// TIA Portal V20 export
// export: Created 2025-12-01T14:57:14.5855708Z, ExportSetting None, DisplayName Totally Integrated Automation Portal, DisplayVersion V20 Update 3, DisplayName TIA Portal Openness, DisplayVersion V20 Update 3, DisplayName TIA Portal Version Control Interface, DisplayVersion V20 Update 3, DisplayName STEP 7 Professional, DisplayVersion V20 Update 3, DisplayName STEP 7 Safety, DisplayVersion V20 Update 2, DisplayName WinCC Basic/Comfort/Advanced, DisplayVersion V20 Update 3, DisplayName WinCC Professional, DisplayVersion V20 Update 3, DisplayName WinCC Unified, DisplayVersion V20 Update 3
FUNCTION "FC700_JDT02ControlTracking" : Void   // FC700, LAD
{ S7_Optimized_Access := 'FALSE' }
AUTHOR : TRACKING
NAME : 20141014
VERSION : 4.0
// stored: AutoNumber false, SetENOAutomatically false
BEGIN

NETWORK
TITLE = Previo
// -----------------------------------------------------------------------
// --- Inicialializacion
// --- Borrado de la Base de Datosç

      CALL  "FC701_JDT02ControlCOM";  // Control del Puerto
      CALL  "FC706_JDT02Borrado";



NETWORK
TITLE = Control del Sistema
// ---------------------------------------------------------------------
// --- Control de Recepcion de Eventos

      CALL  "FC702_JDT02RecJdTMensaje";
      CALL  "FC704_JDT02AnalisisRecibidos";
      CALL  "FC810_EventosRecibidos"
      ( NumJDT := 2
      );


// ---------------------------------------------------------------------
// --- Control de EmisionEventos de Eventos

      CALL  "FC811_EventosGenerados"
      ( NumJdT := 2
      );
      CALL  "FC705_JDT02AnalisisEnviados";
      CALL  "FC703_JDT02EmiJdTMensaje";


// ---------------------------------------------------------------------
// --- Control de EmisionEventos de Router
//     *  Proceso Inicialización bucle
//     *  Eventos de la Pantalla (Movimientos)
//     *  Eventos de Reset V2.0   >>> 2023 01 05

//      CALL  "FC816_EventosEnv_Router"
//         NumJDT :=2

// NIEVES 10/04/25
      CALL  "FC717_Emision_Routing"
      ( NumJDT := 2
      );


      CALL  "FC815_EventosEnv_Control"
      ( NumJDT := 2
      );
      CALL  "FC817_EventosEnv_Reset"
      ( NumJDT := 2
      );


Fin:  NOP   0;


END_FUNCTION
